FUNCTION P2WCHAR : WCHAR
VAR_INPUT
	p : POINTER TO WSTRING;
END_VAR
VAR
END_VAR

P2WCHAR := p^;

END_FUNCTION

(* stored: Version 1.1.0.1, ProductVersion 3.1.4024.11
   POU P2WCHAR: Id {ba926b66-5857-4b56-a633-1867d0a64390}, SpecialFunc None *)
